REGION Network 4: Start injection
   RUNG wire#powerrail
      { S7_Templates := "SrcType := UInt" } EQ_Contact(in1 := #Current_machine_state, in2 := #st_running_molding_sub3)
      wire#w1
      { S7_Templates := "SrcType := UInt" } EQ_Contact(in1 := #Product_no, in2 := 5)
      Move(in := #container_05gr, out1 => #injection_value)
   END_RUNG
   RUNG wire#w1
      { S7_Templates := "SrcType := UInt" } EQ_Contact(in1 := #Product_no, in2 := 1)
      Move(in := #container_1gr, out1 => #injection_value)
   END_RUNG
   RUNG wire#w1
      { S7_Templates := "SrcType := UInt" } EQ_Contact(in1 := #Product_no, in2 := 2)
      Move(in := #container_2gr, out1 => #injection_value)
   END_RUNG
   RUNG wire#w1
      S_Coil( #Injection_start )
   END_RUNG
   RUNG wire#w1
      Contact( #Injection_start )
      { S7_Templates := "SrcType := Real" } LE_Contact(in1 := #injected_value, in2 := #injection_value)
      wire#w2
      { S7_Templates := "SrcType := Real" } Add(in1 := #injected_value, in2 := 1.03, out => #injected_value)
   END_RUNG
   RUNG wire#w2
      Sub(in1 := #Analog_Inputs.Material_ActLevel, in2 := 0.00103, out => #Analog_Inputs.Material_ActLevel)
   END_RUNG
   RUNG wire#w1
      { S7_Templates := "SrcType := Real" } GT_Contact(in1 := #injected_value, in2 := #injection_value)
      wire#w3
      R_Coil( #Injection_start )
   END_RUNG
   RUNG wire#w3
      "FC_change_machineState"(stop_request := #stop_request, new_stateNo := #st_running_molding_sub4, new_stateDescription := 'Waiting for melting', act_error_code := 0, act_warning_code := 0, act_stateNo => #Current_machine_state, info_actStateNo => #StationInfo.StateNo, info_actStateDescription => #StationInfo.StateDescription, info_errorCode => #StationInfo.ErrorCode, info_warningCode => #StationInfo.WarningCode)
   END_RUNG
   // the same network as SCL:
   #_w1 := #Current_machine_state = #st_running_molding_sub3;
   IF #_w1 AND (#Product_no = 5) THEN #injection_value := #container_05gr; END_IF;
   IF #_w1 AND (#Product_no = 1) THEN #injection_value := #container_1gr; END_IF;
   IF #_w1 AND (#Product_no = 2) THEN #injection_value := #container_2gr; END_IF;
   IF #_w1 THEN #Injection_start := TRUE; END_IF;
   #_w2 := #_w1 AND #Injection_start AND (#injected_value <= #injection_value);
   IF #_w2 THEN
       #injected_value := #injected_value + 1.03;
       #Analog_Inputs.Material_ActLevel := #Analog_Inputs.Material_ActLevel - 0.00103;
   END_IF;
   IF #_w1 AND (#injected_value > #injection_value) THEN
       #Injection_start := FALSE;
       "FC_change_machineState"(stop_request := #stop_request,
                               new_stateNo := #st_running_molding_sub4,
                               new_stateDescription := 'Waiting for melting',
                               act_error_code := 0,
                               act_warning_code := 0,
                               act_stateNo => #Current_machine_state,
                               info_actStateNo => #StationInfo.StateNo,
                               info_actStateDescription => #StationInfo.StateDescription,
                               info_errorCode => #StationInfo.ErrorCode,
                               info_warningCode => #StationInfo.WarningCode);
   END_IF;
END_REGION

REGION Network 5
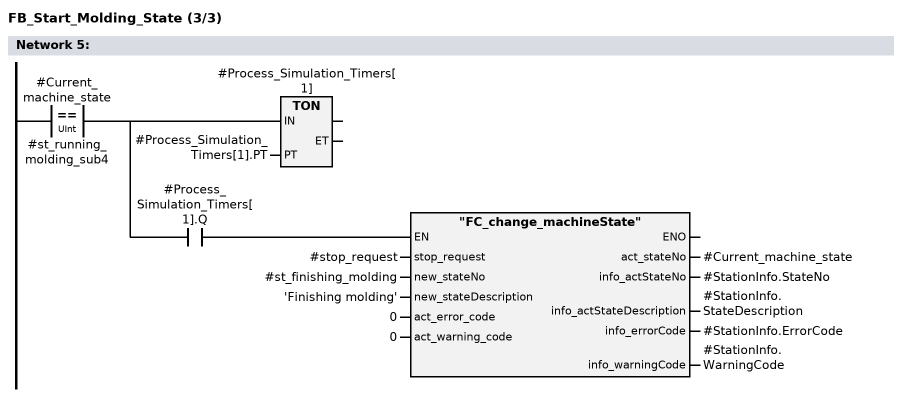
   #_w1 := #Current_machine_state = #st_running_molding_sub4;
   #Process_Simulation_Timers[1].TON(IN := #_w1, PT := #Process_Simulation_Timers[1].PT);
   IF #_w1 AND #Process_Simulation_Timers[1].Q THEN
       "FC_change_machineState"(stop_request := #stop_request,
                               new_stateNo := #st_finishing_molding,
                               new_stateDescription := 'Finishing molding',
                               act_error_code := 0,
                               act_warning_code := 0,
                               act_stateNo => #Current_machine_state,
                               info_actStateNo => #StationInfo.StateNo,
                               info_actStateDescription => #StationInfo.StateDescription,
                               info_errorCode => #StationInfo.ErrorCode,
                               info_warningCode => #StationInfo.WarningCode);
   END_IF;
END_REGION
END_FUNCTION_BLOCK

// folder: Flow4_Finishing_Molding_State

FUNCTION_BLOCK "FB_Finishing_Molding"   // FB12, LAD
{ S7_Optimized_Access := 'TRUE' }
VERSION : 0.1
   VAR_INPUT
      Analog_Inputs : Struct
         Material_ActLevel : Real;
         Temperature_ActLevel : Real;
         Air_Pressure_ActLevel : Real;
         AI_unused1 : Real;
         AI_unused2 : Real;
      END_STRUCT;
      Station_Parameters : Struct
         Hopper : Struct
            ErrorLimit : Real := 1250.0;
            HighLimit : Real := 1000.0;
            LowLimit : Real := 350.0;
            EmptyLimit : Real := 50.0;
         END_STRUCT;
         Temperature : Struct
            ErrorLimit : Real := 600.0;
            HighLimit : Real := 550.0;
            LowLimit : Real := 400.0;
         END_STRUCT;
         Pressure : Struct
            ErrorLimit : Real := 15.0;
            HighLimit : Real := 13.0;
            LowLimit : Real := 10.0;
         END_STRUCT;
         Timeout : Struct
            Mold : Struct
               Open : Time;
               Close : Time;
            END_STRUCT;
            Ejector : Struct
               Open : Time;
               Close : Time;
            END_STRUCT;
            ProductDetect : Time;
            Transfer : Time;
         END_STRUCT;
      END_STRUCT;
   END_VAR
   VAR_OUTPUT
      Ejector_Forward : Bool;
      Ejector_Backward : Bool;
   END_VAR
   VAR_IN_OUT
      Digital_Inputs : Struct
         Start_Button : Bool;
         Stop_Button : Bool;
         Emergency_Stop : Bool;
         Mold_isClosed : Bool;
         Mold_isOpen : Bool;
         Ejector_is_atHome : Bool;
         Ejector_isExtended : Bool;
         Product_Ejected : Bool;
         NextStation_Buffer_Full : Bool;
         DI_unused1 : Bool;
         DI_unused2 : Bool;
         DI_unused3 : Bool;
         DI_unused4 : Bool;
         DI_unused5 : Bool;
         DI_unused6 : Bool;
         DI_unused7 : Bool;
      END_STRUCT;
      stop_request : Bool;
      Current_machine_state : UInt;
      StationInfo : Struct
         StateNo : UInt;
         StateDescription : String;
         ErrorCode : UInt;
         ErrorDescription : String;
         WarningCode : UInt;
         WarninDescription : String;
         TotalProductionTime : Time;
         ProducedCount : UInt;
         OrderCompleted : Bool;
      END_STRUCT;
      Cooler_enable : Bool;
      Mold_open : Bool;
   END_VAR
   VAR
      temp_state : UInt;
      Timeout : Array[0..5] of IEC_TIMER;
      Process_Simulation_Timers : Array[0..20] of IEC_TIMER;
      aux_var1 : Bool;
      deneme_count : IEC_COUNTER;
   END_VAR
   VAR CONSTANT
      st_idle : UInt := 0;
      st_finishing_molding : UInt := 400;
      st_finishing_molding_sub1 : UInt := 401;
      st_finishing_molding_sub2 : UInt := 402;
      st_finishing_molding_sub3 : UInt := 403;
      st_finishing_molding_sub4 : UInt := 404;
      st_finishing_molding_sub5 : UInt := 405;
      st_finishing_molding_sub6 : UInt := 406;
      st_finishing_molding_sub7 : UInt := 407;
      st_finishing_molding_sub8 : UInt := 408;
      st_finishing_molding_sub9 : UInt := 409;
      st_cycle_completed : UInt := 500;
   END_VAR
   VAR_TEMP   // added for the SCL form of the ladder/FBD networks
      _w1 : Bool;
   END_VAR
   // Process_Simulation_Timers[0].PT := T#2S_500MS;
   // Process_Simulation_Timers[1].PT := T#2S_500MS;
   // Process_Simulation_Timers[2].PT := T#500MS;
   // Process_Simulation_Timers[3].PT := T#5S;
   // Process_Simulation_Timers[4].PT := T#10S;
   // Process_Simulation_Timers[10].PT := T#5S;
   // deneme_count.PV := 10;
BEGIN

REGION Network 1
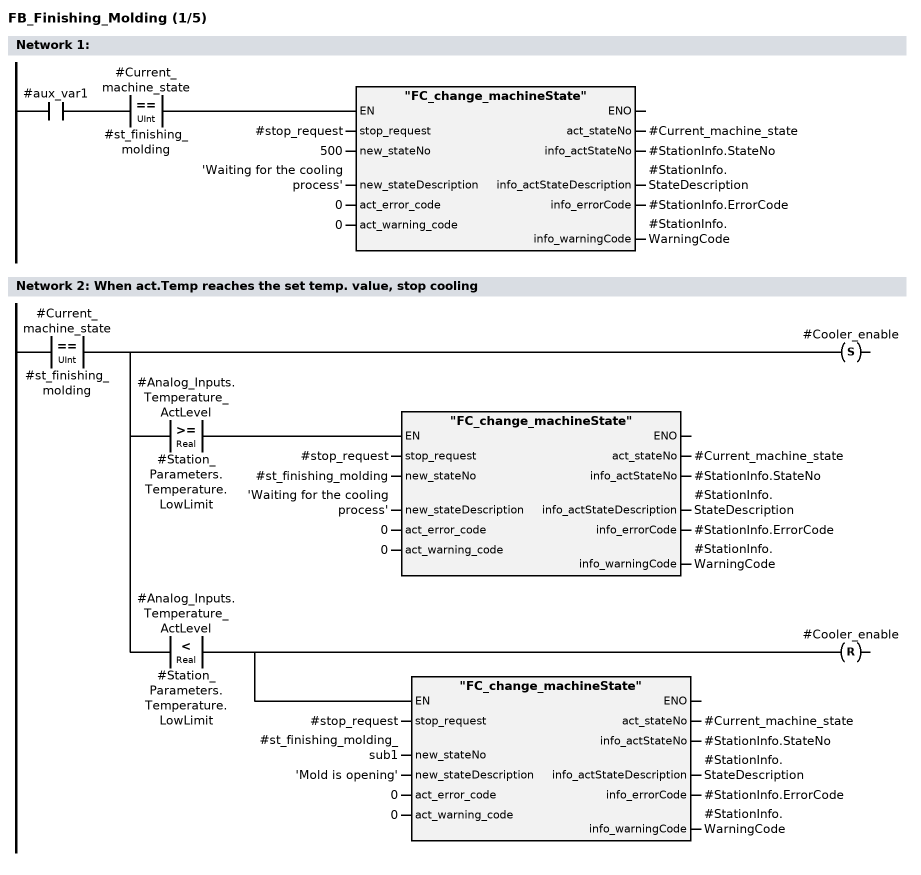
   RUNG wire#powerrail
      Contact( #aux_var1 )
      { S7_Templates := "SrcType := UInt" } EQ_Contact(in1 := #Current_machine_state, in2 := #st_finishing_molding)
      "FC_change_machineState"(stop_request := #stop_request, new_stateNo := 500, new_stateDescription := 'Waiting for the cooling process', act_error_code := 0, act_warning_code := 0, act_stateNo => #Current_machine_state, info_actStateNo => #StationInfo.StateNo, info_actStateDescription => #StationInfo.StateDescription, info_errorCode => #StationInfo.ErrorCode, info_warningCode => #StationInfo.WarningCode)
   END_RUNG
   // the same network as SCL:
   IF #aux_var1 AND (#Current_machine_state = #st_finishing_molding) THEN
       "FC_change_machineState"(stop_request := #stop_request,
                               new_stateNo := 500,
                               new_stateDescription := 'Waiting for the cooling process',
                               act_error_code := 0,
                               act_warning_code := 0,
                               act_stateNo => #Current_machine_state,
                               info_actStateNo => #StationInfo.StateNo,
                               info_actStateDescription => #StationInfo.StateDescription,
                               info_errorCode => #StationInfo.ErrorCode,
                               info_warningCode => #StationInfo.WarningCode);
   END_IF;
END_REGION

REGION Network 2: When act.Temp reaches the set temp. value, stop cooling
   RUNG wire#powerrail
      { S7_Templates := "SrcType := UInt" } EQ_Contact(in1 := #Current_machine_state, in2 := #st_finishing_molding)
      wire#w1
      S_Coil( #Cooler_enable )
   END_RUNG
   RUNG wire#w1
      { S7_Templates := "SrcType := Real" } GE_Contact(in1 := #Analog_Inputs.Temperature_ActLevel, in2 := #Station_Parameters.Temperature.LowLimit)
      "FC_change_machineState"(stop_request := #stop_request, new_stateNo := #st_finishing_molding, new_stateDescription := 'Waiting for the cooling process', act_error_code := 0, act_warning_code := 0, act_stateNo => #Current_machine_state, info_actStateNo => #StationInfo.StateNo, info_actStateDescription => #StationInfo.StateDescription, info_errorCode => #StationInfo.ErrorCode, info_warningCode => #StationInfo.WarningCode)
   END_RUNG
   RUNG wire#w1
      { S7_Templates := "SrcType := Real" } LT_Contact(in1 := #Analog_Inputs.Temperature_ActLevel, in2 := #Station_Parameters.Temperature.LowLimit)
      wire#w2
      R_Coil( #Cooler_enable )
   END_RUNG
   RUNG wire#w2
      "FC_change_machineState"(stop_request := #stop_request, new_stateNo := #st_finishing_molding_sub1, new_stateDescription := 'Mold is opening', act_error_code := 0, act_warning_code := 0, act_stateNo => #Current_machine_state, info_actStateNo => #StationInfo.StateNo, info_actStateDescription => #StationInfo.StateDescription, info_errorCode => #StationInfo.ErrorCode, info_warningCode => #StationInfo.WarningCode)
   END_RUNG
   // the same network as SCL:
   #_w1 := #Current_machine_state = #st_finishing_molding;
   IF #_w1 THEN #Cooler_enable := TRUE; END_IF;
   IF #_w1 AND (#Analog_Inputs.Temperature_ActLevel >= #Station_Parameters.Temperature.LowLimit) THEN
       "FC_change_machineState"(stop_request := #stop_request,
                               new_stateNo := #st_finishing_molding,
                               new_stateDescription := 'Waiting for the cooling process',
                               act_error_code := 0,
                               act_warning_code := 0,
                               act_stateNo => #Current_machine_state,
                               info_actStateNo => #StationInfo.StateNo,
                               info_actStateDescription => #StationInfo.StateDescription,
                               info_errorCode => #StationInfo.ErrorCode,
                               info_warningCode => #StationInfo.WarningCode);
   END_IF;
   IF #_w1 AND (#Analog_Inputs.Temperature_ActLevel < #Station_Parameters.Temperature.LowLimit) THEN
       #Cooler_enable := FALSE;
       "FC_change_machineState"(stop_request := #stop_request,
                               new_stateNo := #st_finishing_molding_sub1,
                               new_stateDescription := 'Mold is opening',
                               act_error_code := 0,
                               act_warning_code := 0,
                               act_stateNo => #Current_machine_state,
                               info_actStateNo => #StationInfo.StateNo,
                               info_actStateDescription => #StationInfo.StateDescription,
                               info_errorCode => #StationInfo.ErrorCode,
                               info_warningCode => #StationInfo.WarningCode);
   END_IF;
END_REGION

REGION Network 3: Open the mold
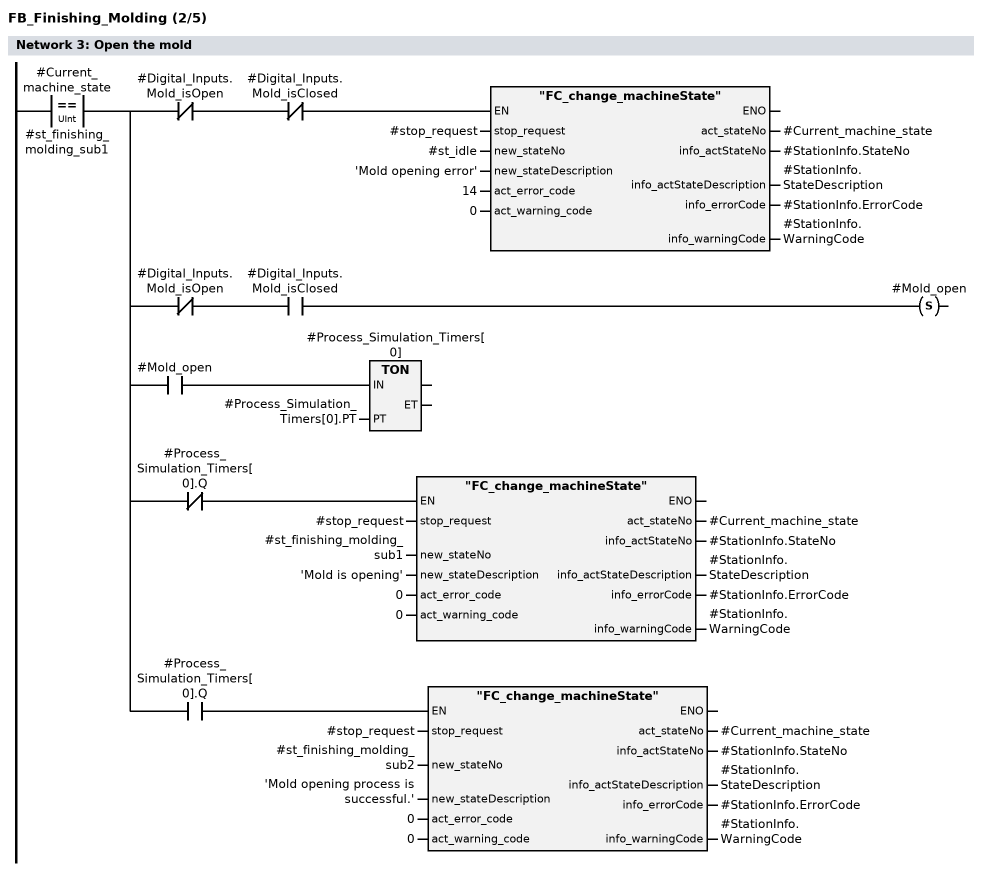
   #_w1 := #Current_machine_state = #st_finishing_molding_sub1;
   IF #_w1 AND NOT #Digital_Inputs.Mold_isOpen AND NOT #Digital_Inputs.Mold_isClosed THEN
       "FC_change_machineState"(stop_request := #stop_request,
                               new_stateNo := #st_idle,
                               new_stateDescription := 'Mold opening error',
                               act_error_code := 14,
                               act_warning_code := 0,
                               act_stateNo => #Current_machine_state,
                               info_actStateNo => #StationInfo.StateNo,
                               info_actStateDescription => #StationInfo.StateDescription,
                               info_errorCode => #StationInfo.ErrorCode,
                               info_warningCode => #StationInfo.WarningCode);
   END_IF;
   IF #_w1 AND NOT #Digital_Inputs.Mold_isOpen AND #Digital_Inputs.Mold_isClosed THEN
       #Mold_open := TRUE;
   END_IF;
   #Process_Simulation_Timers[0].TON(IN := #_w1 AND #Mold_open, PT := #Process_Simulation_Timers[0].PT);
   IF #_w1 AND NOT #Process_Simulation_Timers[0].Q THEN
       "FC_change_machineState"(stop_request := #stop_request,
                               new_stateNo := #st_finishing_molding_sub1,
                               new_stateDescription := 'Mold is opening',
                               act_error_code := 0,
                               act_warning_code := 0,
                               act_stateNo => #Current_machine_state,
                               info_actStateNo => #StationInfo.StateNo,
                               info_actStateDescription => #StationInfo.StateDescription,
                               info_errorCode => #StationInfo.ErrorCode,
                               info_warningCode => #StationInfo.WarningCode);
   END_IF;
   IF #_w1 AND #Process_Simulation_Timers[0].Q THEN
       "FC_change_machineState"(stop_request := #stop_request,
                               new_stateNo := #st_finishing_molding_sub2,
                               new_stateDescription := 'Mold opening process is successful.',
                               act_error_code := 0,
                               act_warning_code := 0,
                               act_stateNo => #Current_machine_state,
                               info_actStateNo => #StationInfo.StateNo,
                               info_actStateDescription => #StationInfo.StateDescription,
                               info_errorCode => #StationInfo.ErrorCode,
                               info_warningCode => #StationInfo.WarningCode);
   END_IF;
END_REGION

REGION Network 4: Start Ejection
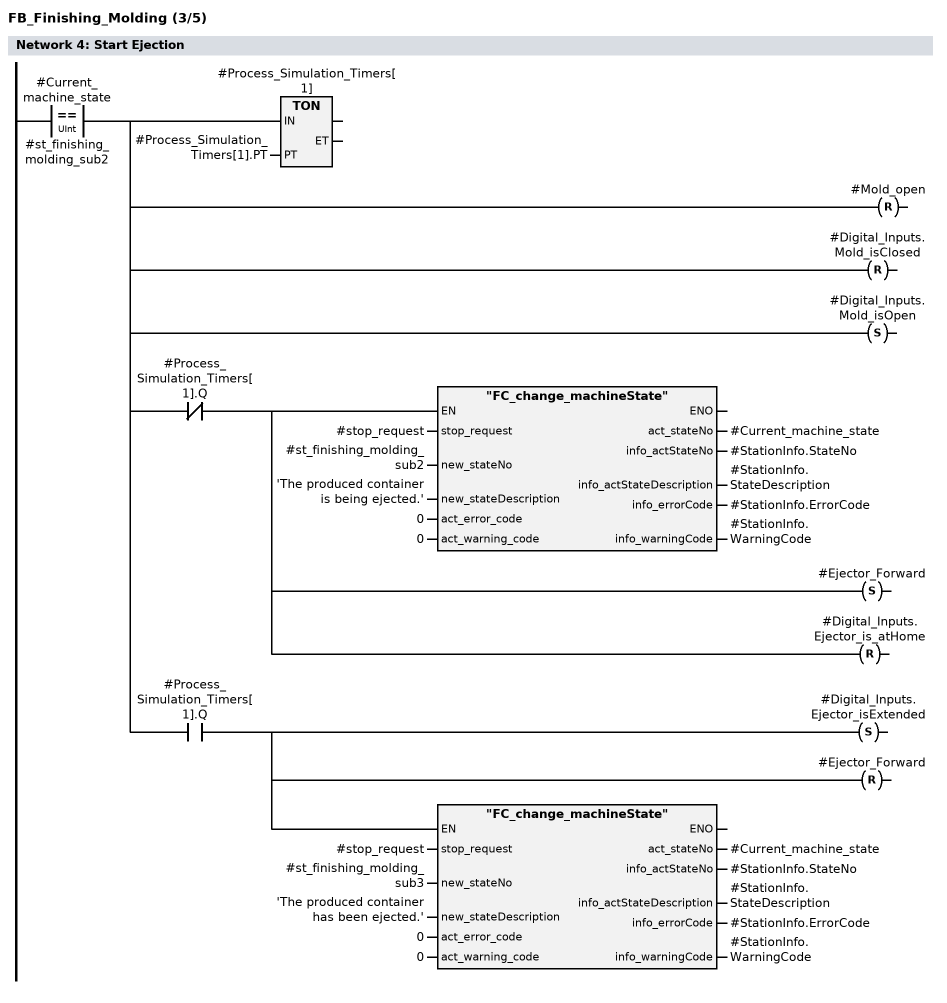
   #_w1 := #Current_machine_state = #st_finishing_molding_sub2;
   #Process_Simulation_Timers[1].TON(IN := #_w1, PT := #Process_Simulation_Timers[1].PT);
   IF #_w1 THEN
       #Mold_open := FALSE;
       #Digital_Inputs.Mold_isClosed := FALSE;
       #Digital_Inputs.Mold_isOpen := TRUE;
   END_IF;
   IF #_w1 AND NOT #Process_Simulation_Timers[1].Q THEN
       "FC_change_machineState"(stop_request := #stop_request,
                               new_stateNo := #st_finishing_molding_sub2,
                               new_stateDescription := 'The produced container is being ejected.',
                               act_error_code := 0,
                               act_warning_code := 0,
                               act_stateNo => #Current_machine_state,
                               info_actStateNo => #StationInfo.StateNo,
                               info_actStateDescription => #StationInfo.StateDescription,
                               info_errorCode => #StationInfo.ErrorCode,
                               info_warningCode => #StationInfo.WarningCode);
       #Ejector_Forward := TRUE;
       #Digital_Inputs.Ejector_is_atHome := FALSE;
   END_IF;
   IF #_w1 AND #Process_Simulation_Timers[1].Q THEN
       #Digital_Inputs.Ejector_isExtended := TRUE;
       #Ejector_Forward := FALSE;
       "FC_change_machineState"(stop_request := #stop_request,
                               new_stateNo := #st_finishing_molding_sub3,
                               new_stateDescription := 'The produced container has been ejected.',
                               act_error_code := 0,
                               act_warning_code := 0,
                               act_stateNo => #Current_machine_state,
                               info_actStateNo => #StationInfo.StateNo,
                               info_actStateDescription => #StationInfo.StateDescription,
                               info_errorCode => #StationInfo.ErrorCode,
                               info_warningCode => #StationInfo.WarningCode);
   END_IF;
END_REGION

REGION Network 5: Stop Ejection
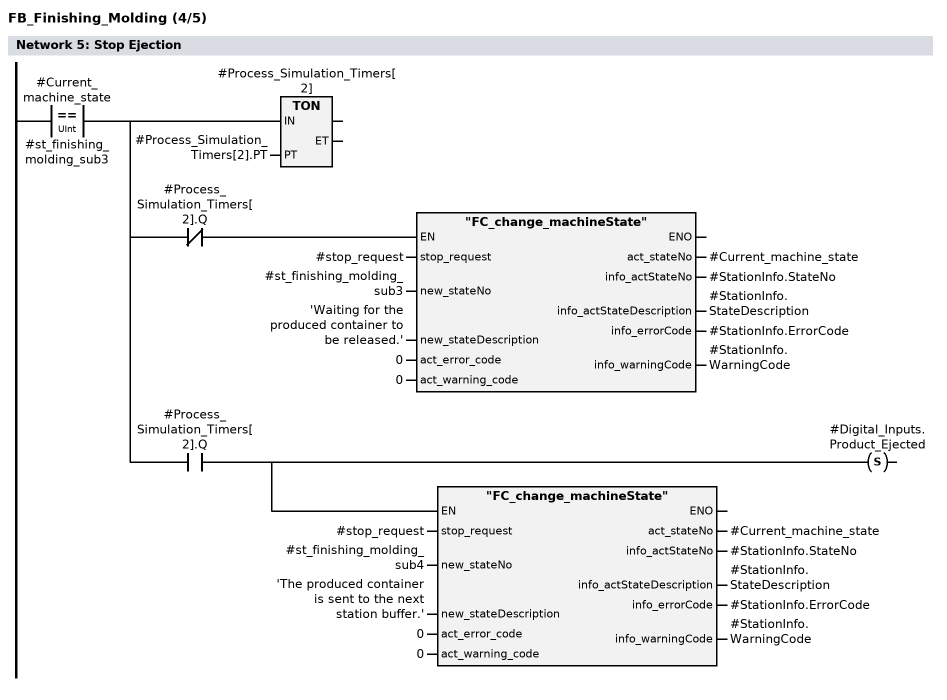
   #_w1 := #Current_machine_state = #st_finishing_molding_sub3;
   #Process_Simulation_Timers[2].TON(IN := #_w1, PT := #Process_Simulation_Timers[2].PT);
   IF #_w1 AND NOT #Process_Simulation_Timers[2].Q THEN
       "FC_change_machineState"(stop_request := #stop_request,
                               new_stateNo := #st_finishing_molding_sub3,
                               new_stateDescription := 'Waiting for the produced container to be released.',
                               act_error_code := 0,
                               act_warning_code := 0,
                               act_stateNo => #Current_machine_state,
                               info_actStateNo => #StationInfo.StateNo,
                               info_actStateDescription => #StationInfo.StateDescription,
                               info_errorCode => #StationInfo.ErrorCode,
                               info_warningCode => #StationInfo.WarningCode);
   END_IF;
   IF #_w1 AND #Process_Simulation_Timers[2].Q THEN
       #Digital_Inputs.Product_Ejected := TRUE;
       "FC_change_machineState"(stop_request := #stop_request,
                               new_stateNo := #st_finishing_molding_sub4,
                               new_stateDescription := 'The produced container is sent to the next station buffer.',
                               act_error_code := 0,
                               act_warning_code := 0,
                               act_stateNo => #Current_machine_state,
                               info_actStateNo => #StationInfo.StateNo,
                               info_actStateDescription => #StationInfo.StateDescription,
                               info_errorCode => #StationInfo.ErrorCode,
                               info_warningCode => #StationInfo.WarningCode);
   END_IF;
END_REGION

REGION Network 6: Send to the next station
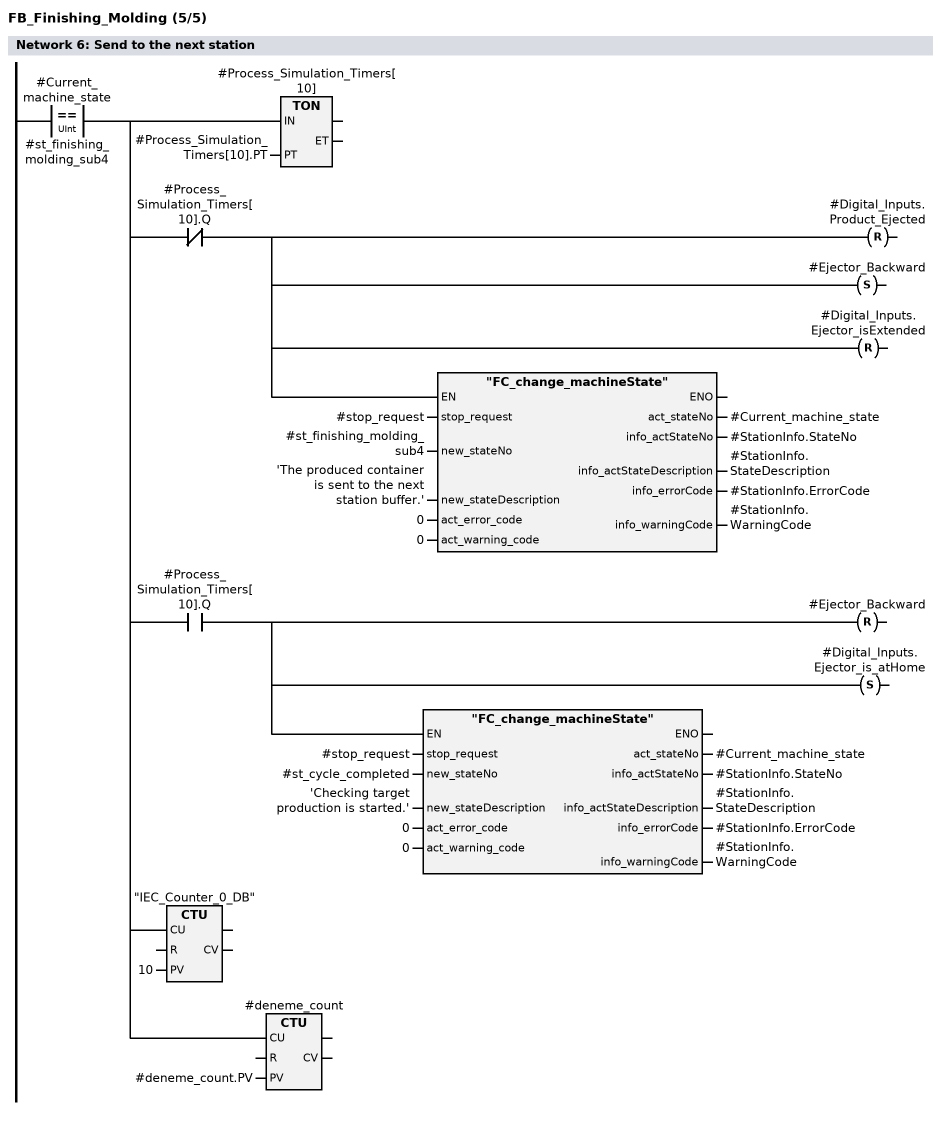
   #_w1 := #Current_machine_state = #st_finishing_molding_sub4;
   #Process_Simulation_Timers[10].TON(IN := #_w1, PT := #Process_Simulation_Timers[10].PT);
   IF #_w1 AND NOT #Process_Simulation_Timers[10].Q THEN
       #Digital_Inputs.Product_Ejected := FALSE;
       #Ejector_Backward := TRUE;
       #Digital_Inputs.Ejector_isExtended := FALSE;
       "FC_change_machineState"(stop_request := #stop_request,
                               new_stateNo := #st_finishing_molding_sub4,
                               new_stateDescription := 'The produced container is sent to the next station buffer.',
                               act_error_code := 0,
                               act_warning_code := 0,
                               act_stateNo => #Current_machine_state,
                               info_actStateNo => #StationInfo.StateNo,
                               info_actStateDescription => #StationInfo.StateDescription,
                               info_errorCode => #StationInfo.ErrorCode,
                               info_warningCode => #StationInfo.WarningCode);
   END_IF;
   IF #_w1 AND #Process_Simulation_Timers[10].Q THEN
       #Ejector_Backward := FALSE;
       #Digital_Inputs.Ejector_is_atHome := TRUE;
       "FC_change_machineState"(stop_request := #stop_request,
                               new_stateNo := #st_cycle_completed,
                               new_stateDescription := 'Checking target production is started.',
                               act_error_code := 0,
                               act_warning_code := 0,
                               act_stateNo => #Current_machine_state,
                               info_actStateNo => #StationInfo.StateNo,
                               info_actStateDescription => #StationInfo.StateDescription,
                               info_errorCode => #StationInfo.ErrorCode,
                               info_warningCode => #StationInfo.WarningCode);
   END_IF;
   "IEC_Counter_0_DB".CTU(CU := #_w1, PV := 10);
   #deneme_count.CTU(CU := #_w1, PV := #deneme_count.PV);
END_REGION
END_FUNCTION_BLOCK

// folder: Flow5_Checking_Target_Production

FUNCTION_BLOCK "FB_Checking_Target_Production"   // FB11, LAD
{ S7_Optimized_Access := 'TRUE' }
VERSION : 0.1
   VAR_INPUT
      target_quantity : UInt;
   END_VAR
   VAR_IN_OUT
      stop_request : Bool;
      Current_machine_state : UInt;
      StationInfo : Struct
         StateNo : UInt;
         StateDescription : String;
         ErrorCode : UInt;
         ErrorDescription : String;
         WarningCode : UInt;
         WarninDescription : String;
         TotalProductionTime : Time;
         ProducedCount : UInt;
         OrderCompleted : Bool;
      END_STRUCT;
   END_VAR
   VAR
      Timeout : Array[0..5] of IEC_TIMER;
      Process_Simulation_Timers : Array[0..20] of IEC_TIMER;
      Production_Counter : Array[0..10] of IEC_UCOUNTER;
      aux_var1 : Bool;
   END_VAR
   VAR_TEMP
      cycle_completed : Bool;
      continue : Bool;
   END_VAR
   VAR CONSTANT
      st_idle : UInt := 0;
      st_cycle_completed : UInt := 500;
      st_cycle_completed_sub1 : UInt := 501;
      st_cycle_completed_sub2 : UInt := 502;
      st_cycle_completed_sub3 : UInt := 503;
      st_cycle_completed_sub4 : UInt := 504;
      st_cycle_completed_sub5 : UInt := 505;
      st_cycle_completed_sub6 : UInt := 506;
      st_cycle_completed_sub7 : UInt := 507;
      st_cycle_completed_sub8 : UInt := 508;
      st_cycle_completed_sub9 : UInt := 509;
      st_checking_order_target : UInt := 600;
      st_checking_initial_safety : UInt := 200;
      st_order_finishing : UInt := 700;
      st_checking_order_sub2 : UInt := 102;
   END_VAR
   VAR_TEMP   // added for the SCL form of the ladder/FBD networks
      _w1 : Bool;
   END_VAR
   // Process_Simulation_Timers[0].PT := T#3S;
   // Process_Simulation_Timers[1].PT := T#4S;
   // Process_Simulation_Timers[2].PT := T#10S;
   // Process_Simulation_Timers[3].PT := T#3S;
BEGIN

REGION Network 1: Check target production
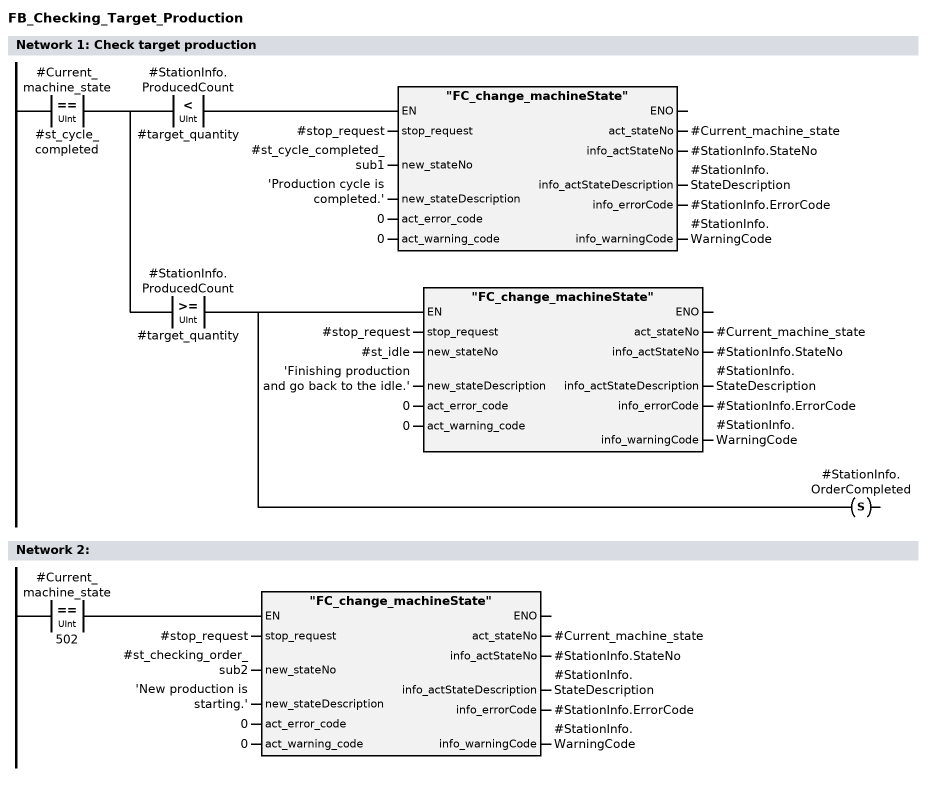
   RUNG wire#powerrail
      { S7_Templates := "SrcType := UInt" } EQ_Contact(in1 := #Current_machine_state, in2 := #st_cycle_completed)
      wire#w1
      { S7_Templates := "SrcType := UInt" } LT_Contact(in1 := #StationInfo.ProducedCount, in2 := #target_quantity)
      "FC_change_machineState"(stop_request := #stop_request, new_stateNo := #st_cycle_completed_sub1, new_stateDescription := 'Production cycle is completed.', act_error_code := 0, act_warning_code := 0, act_stateNo => #Current_machine_state, info_actStateNo => #StationInfo.StateNo, info_actStateDescription => #StationInfo.StateDescription, info_errorCode => #StationInfo.ErrorCode, info_warningCode => #StationInfo.WarningCode)
   END_RUNG
   RUNG wire#w1
      { S7_Templates := "SrcType := UInt" } GE_Contact(in1 := #StationInfo.ProducedCount, in2 := #target_quantity)
      wire#w2
      "FC_change_machineState"(stop_request := #stop_request, new_stateNo := #st_idle, new_stateDescription := 'Finishing production and go back to the idle.', act_error_code := 0, act_warning_code := 0, act_stateNo => #Current_machine_state, info_actStateNo => #StationInfo.StateNo, info_actStateDescription => #StationInfo.StateDescription, info_errorCode => #StationInfo.ErrorCode, info_warningCode => #StationInfo.WarningCode)
   END_RUNG
   RUNG wire#w2
      S_Coil( #StationInfo.OrderCompleted )
   END_RUNG
   // the same network as SCL:
   #_w1 := #Current_machine_state = #st_cycle_completed;
   IF #_w1 AND (#StationInfo.ProducedCount < #target_quantity) THEN
       "FC_change_machineState"(stop_request := #stop_request,
                               new_stateNo := #st_cycle_completed_sub1,
                               new_stateDescription := 'Production cycle is completed.',
                               act_error_code := 0,
                               act_warning_code := 0,
                               act_stateNo => #Current_machine_state,
                               info_actStateNo => #StationInfo.StateNo,
                               info_actStateDescription => #StationInfo.StateDescription,
                               info_errorCode => #StationInfo.ErrorCode,
                               info_warningCode => #StationInfo.WarningCode);
   END_IF;
   IF #_w1 AND (#StationInfo.ProducedCount >= #target_quantity) THEN
       "FC_change_machineState"(stop_request := #stop_request,
                               new_stateNo := #st_idle,
                               new_stateDescription := 'Finishing production and go back to the idle.',
                               act_error_code := 0,
                               act_warning_code := 0,
                               act_stateNo => #Current_machine_state,
                               info_actStateNo => #StationInfo.StateNo,
                               info_actStateDescription => #StationInfo.StateDescription,
                               info_errorCode => #StationInfo.ErrorCode,
                               info_warningCode => #StationInfo.WarningCode);
       #StationInfo.OrderCompleted := TRUE;
   END_IF;
END_REGION

REGION Network 2
   RUNG wire#powerrail
      { S7_Templates := "SrcType := UInt" } EQ_Contact(in1 := #Current_machine_state, in2 := 502)
      "FC_change_machineState"(stop_request := #stop_request, new_stateNo := #st_checking_order_sub2, new_stateDescription := 'New production is starting.', act_error_code := 0, act_warning_code := 0, act_stateNo => #Current_machine_state, info_actStateNo => #StationInfo.StateNo, info_actStateDescription => #StationInfo.StateDescription, info_errorCode => #StationInfo.ErrorCode, info_warningCode => #StationInfo.WarningCode)
   END_RUNG
   // the same network as SCL:
   IF #Current_machine_state = 502 THEN
       "FC_change_machineState"(stop_request := #stop_request,
                               new_stateNo := #st_checking_order_sub2,
                               new_stateDescription := 'New production is starting.',
                               act_error_code := 0,
                               act_warning_code := 0,
                               act_stateNo => #Current_machine_state,
                               info_actStateNo => #StationInfo.StateNo,
                               info_actStateDescription => #StationInfo.StateDescription,
                               info_errorCode => #StationInfo.ErrorCode,
                               info_warningCode => #StationInfo.WarningCode);
   END_IF;
END_REGION
END_FUNCTION_BLOCK

// folder: Functions

FUNCTION "FC_get_time_data" : Void   // FC1, LAD
{ S7_Optimized_Access := 'TRUE' }
VERSION : 0.1
   VAR_OUTPUT
      actYear : UInt;
      actMonth : UInt;
      actDay : UInt;
      timeStamp : UDInt;
      errorGettingTime : Int;
   END_VAR
   VAR_TEMP
      timeData : DTL;
      gettingTimeState : Int;
   END_VAR
BEGIN

REGION Network 1
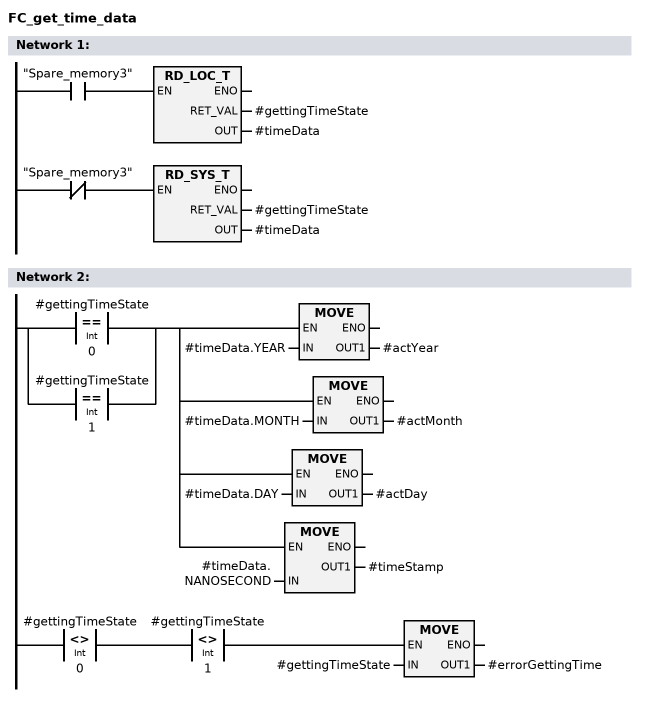
   IF "Spare_memory3" THEN #gettingTimeState := RD_LOC_T(OUT => #timeData); END_IF;
   IF NOT "Spare_memory3" THEN #gettingTimeState := RD_SYS_T(OUT => #timeData); END_IF;
END_REGION

REGION Network 2
   RUNG wire#powerrail
      { S7_Templates := "SrcType := Int" } EQ_Contact(in1 := #gettingTimeState, in2 := 0)
      wire#w1
      Move(in := #timeData.YEAR, out1 => #actYear)
   END_RUNG
   RUNG wire#powerrail
      { S7_Templates := "SrcType := Int" } EQ_Contact(in1 := #gettingTimeState, in2 := 1)
   END_RUNG wire#w1
   RUNG wire#w1
      Move(in := #timeData.MONTH, out1 => #actMonth)
   END_RUNG
   RUNG wire#w1
      Move(in := #timeData.DAY, out1 => #actDay)
   END_RUNG
   RUNG wire#w1
      Move(in := #timeData.NANOSECOND, out1 => #timeStamp)
   END_RUNG
   RUNG wire#powerrail
      { S7_Templates := "SrcType := Int" } NE_Contact(in1 := #gettingTimeState, in2 := 0)
      { S7_Templates := "SrcType := Int" } NE_Contact(in1 := #gettingTimeState, in2 := 1)
      Move(in := #gettingTimeState, out1 => #errorGettingTime)
   END_RUNG
   // the same network as SCL:
   IF (#gettingTimeState = 0) OR (#gettingTimeState = 1) THEN
       #actYear := #timeData.YEAR;
       #actMonth := #timeData.MONTH;
       #actDay := #timeData.DAY;
       #timeStamp := #timeData.NANOSECOND;
   END_IF;
   IF (#gettingTimeState <> 0) AND (#gettingTimeState <> 1) THEN
       #errorGettingTime := #gettingTimeState;
   END_IF;
END_REGION
END_FUNCTION

FUNCTION "FC_change_machineState" : Void   // FC2, LAD
{ S7_Optimized_Access := 'TRUE' }
VERSION : 0.1
   VAR_INPUT
      stop_request : Bool;
      new_stateNo : UInt;
      new_stateDescription : String;
      act_error_code : UInt;
      act_warning_code : UInt;
   END_VAR
   VAR_OUTPUT
      act_stateNo : UInt;
      info_actStateNo : UInt;
      info_actStateDescription : String;
      info_errorCode : UInt;
      info_warningCode : UInt;
   END_VAR
   VAR CONSTANT
      st_idle : UInt := 0;
   END_VAR
BEGIN

REGION Network 1: No Stop Request Received
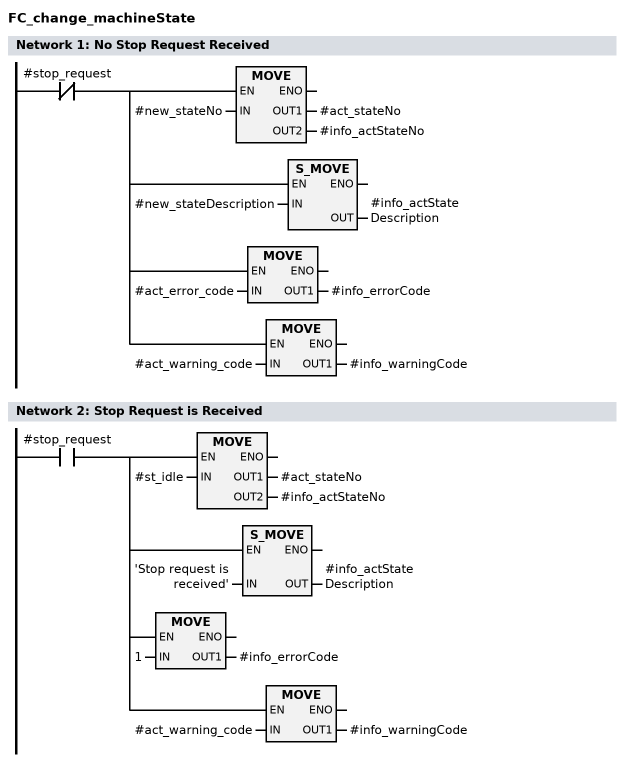
   RUNG wire#powerrail
      I_Contact( #stop_request )
      wire#w1
      Move(in := #new_stateNo, out1 => #act_stateNo, out2 => #info_actStateNo)
   END_RUNG
   RUNG wire#w1
      S_Move(in := #new_stateDescription, out => #info_actStateDescription)
   END_RUNG
   RUNG wire#w1
      Move(in := #act_error_code, out1 => #info_errorCode)
   END_RUNG
   RUNG wire#w1
      Move(in := #act_warning_code, out1 => #info_warningCode)
   END_RUNG
   // the same network as SCL:
   IF NOT #stop_request THEN
       #act_stateNo := #new_stateNo;
       #info_actStateNo := #new_stateNo;
       #info_actStateDescription := #new_stateDescription;
       #info_errorCode := #act_error_code;
       #info_warningCode := #act_warning_code;
   END_IF;
END_REGION

REGION Network 2: Stop Request is Received
   RUNG wire#powerrail
      Contact( #stop_request )
      wire#w1
      Move(in := #st_idle, out1 => #act_stateNo, out2 => #info_actStateNo)
   END_RUNG
   RUNG wire#w1
      S_Move(in := 'Stop request is received', out => #info_actStateDescription)
   END_RUNG
   RUNG wire#w1
      Move(in := 1, out1 => #info_errorCode)
   END_RUNG
   RUNG wire#w1
      Move(in := #act_warning_code, out1 => #info_warningCode)
   END_RUNG
   // the same network as SCL:
   IF #stop_request THEN
       #act_stateNo := #st_idle;
       #info_actStateNo := #st_idle;
       #info_actStateDescription := 'Stop request is received';
       #info_errorCode := 1;
       #info_warningCode := #act_warning_code;
   END_IF;
END_REGION
END_FUNCTION

// folder: Machine_transition

FUNCTION_BLOCK "FB_SubTransition"   // FB3, LAD
{ S7_Optimized_Access := 'TRUE' }
VERSION : 0.1
   VAR_INPUT
      new_state : UInt;
   END_VAR
   VAR_OUTPUT
      new_machine_state : UInt;
      previous_state_done : Bool;
   END_VAR
   VAR_IN_OUT
      stop_request : Bool;
   END_VAR
   VAR CONSTANT
      st_idle : UInt := 0;
   END_VAR
BEGIN

REGION Network 1: No Stop Request
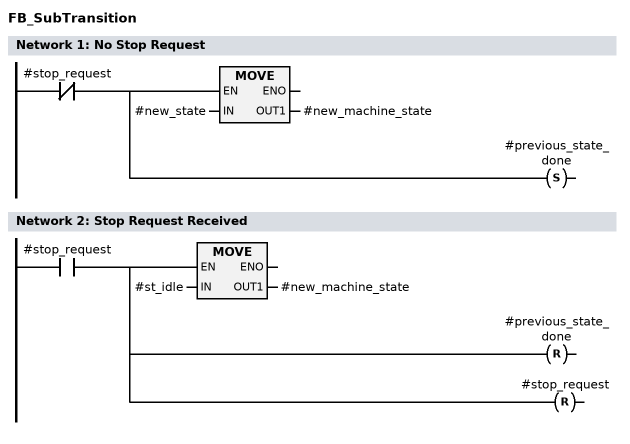
   RUNG wire#powerrail
      I_Contact( #stop_request )
      wire#w1
      Move(in := #new_state, out1 => #new_machine_state)
   END_RUNG
   RUNG wire#w1
      S_Coil( #previous_state_done )
   END_RUNG
   // the same network as SCL:
   IF NOT #stop_request THEN
       #new_machine_state := #new_state;
       #previous_state_done := TRUE;
   END_IF;
END_REGION

REGION Network 2: Stop Request Received
   RUNG wire#powerrail
      Contact( #stop_request )
      wire#w1
      Move(in := #st_idle, out1 => #new_machine_state)
   END_RUNG
   RUNG wire#w1
      R_Coil( #previous_state_done )
   END_RUNG
   RUNG wire#w1
      R_Coil( #stop_request )
   END_RUNG
   // the same network as SCL:
   IF #stop_request THEN
       #new_machine_state := #st_idle;
       #previous_state_done := FALSE;
       #stop_request := FALSE;
   END_IF;
END_REGION
END_FUNCTION_BLOCK

FUNCTION_BLOCK "FB_control_state_transition"   // FB6, LAD
TITLE = This FB sets the machine status
{ S7_Optimized_Access := 'TRUE' }
VERSION : 0.1
   VAR_INPUT
      is_start_btn_activated : Bool;
      is_stop_btn_activated : Bool;
   END_VAR
   VAR_IN_OUT
      current_machine_state : UInt;
      is_previous_state_done : Bool;
   END_VAR
   VAR
      temp_state : UInt;
      initial_temp_state : UInt;
      stop_request : Bool;
   END_VAR
   VAR CONSTANT
      st_idle : UInt := 0;
      st_checking_order : UInt := 10;
      st_checking_initial_safety : UInt := 20;
      st_checking_material_level : UInt := 30;
      st_running_molding : UInt := 40;
      st_finishing_molding : UInt := 50;
      st_cycle_completed : UInt := 60;
      st_checking_order_target : UInt := 70;
      st_order_finishing : UInt := 80;
      st_fault : UInt := 300;
   END_VAR
   VAR_TEMP   // added for the SCL form of the ladder/FBD networks
      _w1 : Bool;
   END_VAR
BEGIN

REGION Network 1: Control Stop Request
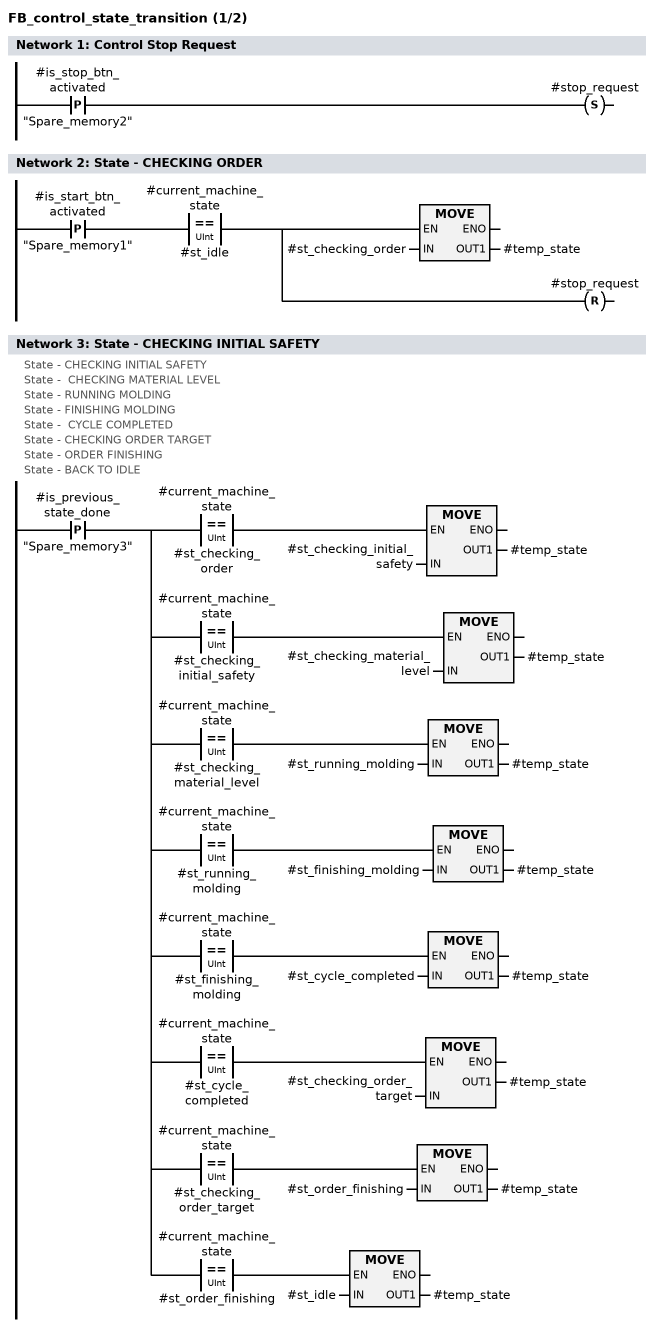
   RUNG wire#powerrail
      P_Contact(operand := #is_stop_btn_activated, bit := "Spare_memory2")
      S_Coil( #stop_request )
   END_RUNG
   // the same network as SCL:
   #_w1 := #is_stop_btn_activated AND NOT "Spare_memory2";   // rising edge of #is_stop_btn_activated
   "Spare_memory2" := #is_stop_btn_activated;
   IF #_w1 THEN #stop_request := TRUE; END_IF;
END_REGION

REGION Network 2: State - CHECKING ORDER
   RUNG wire#powerrail
      P_Contact(operand := #is_start_btn_activated, bit := "Spare_memory1")
      { S7_Templates := "SrcType := UInt" } EQ_Contact(in1 := #current_machine_state, in2 := #st_idle)
      wire#w1
      Move(in := #st_checking_order, out1 => #temp_state)
   END_RUNG
   RUNG wire#w1
      R_Coil( #stop_request )
   END_RUNG
   // the same network as SCL:
   #_w1 := #is_start_btn_activated AND NOT "Spare_memory1";   // rising edge of #is_start_btn_activated
   "Spare_memory1" := #is_start_btn_activated;
   IF #_w1 AND (#current_machine_state = #st_idle) THEN
       #temp_state := #st_checking_order;
       #stop_request := FALSE;
   END_IF;
END_REGION

REGION Network 3: State - CHECKING INITIAL SAFETY
   // State - CHECKING INITIAL SAFETY
   // State -  CHECKING MATERIAL LEVEL
   // State - RUNNING MOLDING
   // State - FINISHING MOLDING
   // State -  CYCLE COMPLETED
   // State - CHECKING ORDER TARGET
   // State - ORDER FINISHING 
   // State - BACK TO IDLE
   RUNG wire#powerrail
      P_Contact(operand := #is_previous_state_done, bit := "Spare_memory3")
      wire#w1
      { S7_Templates := "SrcType := UInt" } EQ_Contact(in1 := #current_machine_state, in2 := #st_checking_order)
      Move(in := #st_checking_initial_safety, out1 => #temp_state)
   END_RUNG
   RUNG wire#w1
      { S7_Templates := "SrcType := UInt" } EQ_Contact(in1 := #current_machine_state, in2 := #st_checking_initial_safety)
      Move(in := #st_checking_material_level, out1 => #temp_state)
   END_RUNG
   RUNG wire#w1
      { S7_Templates := "SrcType := UInt" } EQ_Contact(in1 := #current_machine_state, in2 := #st_checking_material_level)
      Move(in := #st_running_molding, out1 => #temp_state)
   END_RUNG
   RUNG wire#w1
      { S7_Templates := "SrcType := UInt" } EQ_Contact(in1 := #current_machine_state, in2 := #st_running_molding)
      Move(in := #st_finishing_molding, out1 => #temp_state)
   END_RUNG
   RUNG wire#w1
      { S7_Templates := "SrcType := UInt" } EQ_Contact(in1 := #current_machine_state, in2 := #st_finishing_molding)
      Move(in := #st_cycle_completed, out1 => #temp_state)
   END_RUNG
   RUNG wire#w1
      { S7_Templates := "SrcType := UInt" } EQ_Contact(in1 := #current_machine_state, in2 := #st_cycle_completed)
      Move(in := #st_checking_order_target, out1 => #temp_state)
   END_RUNG
   RUNG wire#w1
      { S7_Templates := "SrcType := UInt" } EQ_Contact(in1 := #current_machine_state, in2 := #st_checking_order_target)
      Move(in := #st_order_finishing, out1 => #temp_state)
   END_RUNG
   RUNG wire#w1
      { S7_Templates := "SrcType := UInt" } EQ_Contact(in1 := #current_machine_state, in2 := #st_order_finishing)
      Move(in := #st_idle, out1 => #temp_state)
   END_RUNG
   // the same network as SCL:
   #_w1 := #is_previous_state_done AND NOT "Spare_memory3";   // rising edge of #is_previous_state_done
   "Spare_memory3" := #is_previous_state_done;
   IF #_w1 AND (#current_machine_state = #st_checking_order) THEN
       #temp_state := #st_checking_initial_safety;
   END_IF;
   IF #_w1 AND (#current_machine_state = #st_checking_initial_safety) THEN
       #temp_state := #st_checking_material_level;
   END_IF;
   IF #_w1 AND (#current_machine_state = #st_checking_material_level) THEN
       #temp_state := #st_running_molding;
   END_IF;
   IF #_w1 AND (#current_machine_state = #st_running_molding) THEN
       #temp_state := #st_finishing_molding;
   END_IF;
   IF #_w1 AND (#current_machine_state = #st_finishing_molding) THEN
       #temp_state := #st_cycle_completed;
   END_IF;
   IF #_w1 AND (#current_machine_state = #st_cycle_completed) THEN
       #temp_state := #st_checking_order_target;
   END_IF;
   IF #_w1 AND (#current_machine_state = #st_checking_order_target) THEN
       #temp_state := #st_order_finishing;
   END_IF;
   IF #_w1 AND (#current_machine_state = #st_order_finishing) THEN #temp_state := #st_idle; END_IF;
END_REGION

REGION Network 4: Set the current machine state to new state value
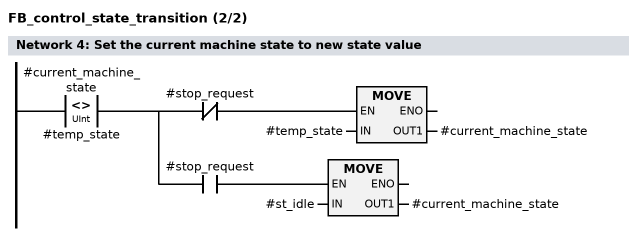
   RUNG wire#powerrail
      { S7_Templates := "SrcType := UInt" } NE_Contact(in1 := #current_machine_state, in2 := #temp_state)
      wire#w1
      I_Contact( #stop_request )
      Move(in := #temp_state, out1 => #current_machine_state)
   END_RUNG
   RUNG wire#w1
      Contact( #stop_request )
      Move(in := #st_idle, out1 => #current_machine_state)
   END_RUNG
   // the same network as SCL:
   #_w1 := #current_machine_state <> #temp_state;
   IF #_w1 AND NOT #stop_request THEN #current_machine_state := #temp_state; END_IF;
   IF #_w1 AND #stop_request THEN #current_machine_state := #st_idle; END_IF;
END_REGION
END_FUNCTION_BLOCK

// folder: Manage_outputs

FUNCTION_BLOCK "FB_manage_outputs"   // FB8, LAD
{ S7_Optimized_Access := 'TRUE' }
VERSION : 0.1
BEGIN

REGION Network 1: Feeder_Start
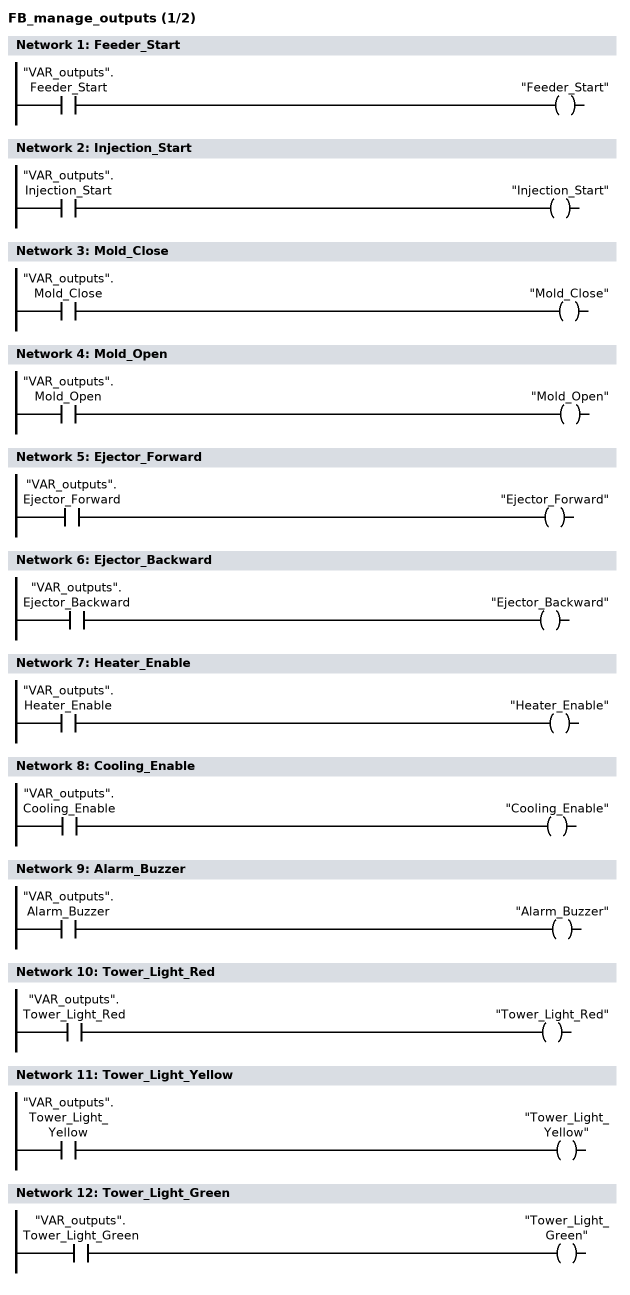
   RUNG wire#powerrail
      Contact( "VAR_outputs".Feeder_Start )
      Coil( "Feeder_Start" )
   END_RUNG
   // the same network as SCL:
   "Feeder_Start" := "VAR_outputs".Feeder_Start;
END_REGION

REGION Network 2: Injection_Start
   RUNG wire#powerrail
      Contact( "VAR_outputs".Injection_Start )
      Coil( "Injection_Start" )
   END_RUNG
   // the same network as SCL:
   "Injection_Start" := "VAR_outputs".Injection_Start;
END_REGION

REGION Network 3: Mold_Close
   RUNG wire#powerrail
      Contact( "VAR_outputs".Mold_Close )
      Coil( "Mold_Close" )
   END_RUNG
   // the same network as SCL:
   "Mold_Close" := "VAR_outputs".Mold_Close;
END_REGION

REGION Network 4: Mold_Open
   RUNG wire#powerrail
      Contact( "VAR_outputs".Mold_Open )
      Coil( "Mold_Open" )
   END_RUNG
   // the same network as SCL:
   "Mold_Open" := "VAR_outputs".Mold_Open;
END_REGION

REGION Network 5: Ejector_Forward
   RUNG wire#powerrail
      Contact( "VAR_outputs".Ejector_Forward )
      Coil( "Ejector_Forward" )
   END_RUNG
   // the same network as SCL:
   "Ejector_Forward" := "VAR_outputs".Ejector_Forward;
END_REGION

REGION Network 6: Ejector_Backward
   RUNG wire#powerrail
      Contact( "VAR_outputs".Ejector_Backward )
      Coil( "Ejector_Backward" )
   END_RUNG
   // the same network as SCL:
   "Ejector_Backward" := "VAR_outputs".Ejector_Backward;
END_REGION

REGION Network 7: Heater_Enable
   RUNG wire#powerrail
      Contact( "VAR_outputs".Heater_Enable )
      Coil( "Heater_Enable" )
   END_RUNG
   // the same network as SCL:
   "Heater_Enable" := "VAR_outputs".Heater_Enable;
END_REGION

REGION Network 8: Cooling_Enable
   RUNG wire#powerrail
      Contact( "VAR_outputs".Cooling_Enable )
      Coil( "Cooling_Enable" )
   END_RUNG
   // the same network as SCL:
   "Cooling_Enable" := "VAR_outputs".Cooling_Enable;
END_REGION

REGION Network 9: Alarm_Buzzer
   RUNG wire#powerrail
      Contact( "VAR_outputs".Alarm_Buzzer )
      Coil( "Alarm_Buzzer" )
   END_RUNG
   // the same network as SCL:
   "Alarm_Buzzer" := "VAR_outputs".Alarm_Buzzer;
END_REGION

REGION Network 10: Tower_Light_Red
   RUNG wire#powerrail
      Contact( "VAR_outputs".Tower_Light_Red )
      Coil( "Tower_Light_Red" )
   END_RUNG
   // the same network as SCL:
   "Tower_Light_Red" := "VAR_outputs".Tower_Light_Red;
END_REGION

REGION Network 11: Tower_Light_Yellow
   RUNG wire#powerrail
      Contact( "VAR_outputs".Tower_Light_Yellow )
      Coil( "Tower_Light_Yellow" )
   END_RUNG
   // the same network as SCL:
   "Tower_Light_Yellow" := "VAR_outputs".Tower_Light_Yellow;
END_REGION

REGION Network 12: Tower_Light_Green
   RUNG wire#powerrail
      Contact( "VAR_outputs".Tower_Light_Green )
      Coil( "Tower_Light_Green" )
   END_RUNG
   // the same network as SCL:
   "Tower_Light_Green" := "VAR_outputs".Tower_Light_Green;
END_REGION

REGION Network 13: Goto_NextStationBuffer
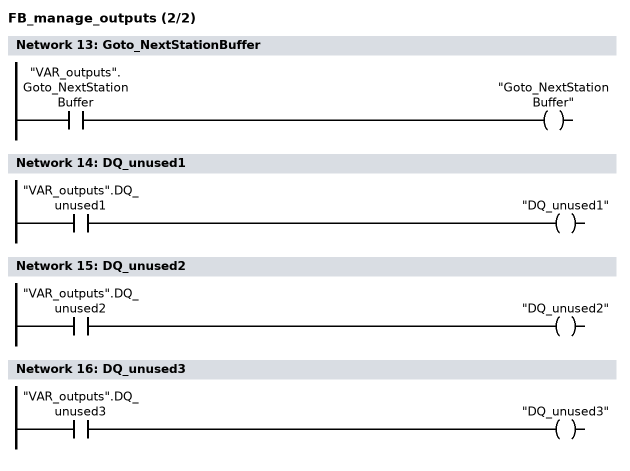
   RUNG wire#powerrail
      Contact( "VAR_outputs".Goto_NextStationBuffer )
      Coil( "Goto_NextStationBuffer" )
   END_RUNG
   // the same network as SCL:
   "Goto_NextStationBuffer" := "VAR_outputs".Goto_NextStationBuffer;
END_REGION

REGION Network 14: DQ_unused1
   RUNG wire#powerrail
      Contact( "VAR_outputs".DQ_unused1 )
      Coil( "DQ_unused1" )
   END_RUNG
   // the same network as SCL:
   "DQ_unused1" := "VAR_outputs".DQ_unused1;
END_REGION

REGION Network 15: DQ_unused2
   RUNG wire#powerrail
      Contact( "VAR_outputs".DQ_unused2 )
      Coil( "DQ_unused2" )
   END_RUNG
   // the same network as SCL:
   "DQ_unused2" := "VAR_outputs".DQ_unused2;
END_REGION

REGION Network 16: DQ_unused3
   RUNG wire#powerrail
      Contact( "VAR_outputs".DQ_unused3 )
      Coil( "DQ_unused3" )
   END_RUNG
   // the same network as SCL:
   "DQ_unused3" := "VAR_outputs".DQ_unused3;
END_REGION
END_FUNCTION_BLOCK

// folder: Simulation_data/Simulation_FB

FUNCTION_BLOCK "FB_simulate_analog_data"   // FB10, LAD
{ S7_Optimized_Access := 'TRUE' }
VERSION : 0.1
   VAR_INPUT
      Clock : Bool;
      Up : Bool;
      Down : Bool;
      TargetLevelLimit : Real;
      HighLevelLimit : Real;
      LowLevelLimit : Real;
      ResetVal : Bool;
   END_VAR
   VAR_IN_OUT
      actLevel : Real;
   END_VAR
   VAR
      value_int : Int;
      value_real : Real;
   END_VAR
   VAR_TEMP
      tag1 : Bool;
   END_VAR
   VAR CONSTANT
      incrementVal : Int := 5;
      decrementVal : Int := 150;
      normMin : Int := 0;
      normMax : Int := 27648;
   END_VAR
   VAR_TEMP   // added for the SCL form of the ladder/FBD networks
      _w1 : Bool;
   END_VAR
BEGIN

REGION Network 1: Simulate an analog input value
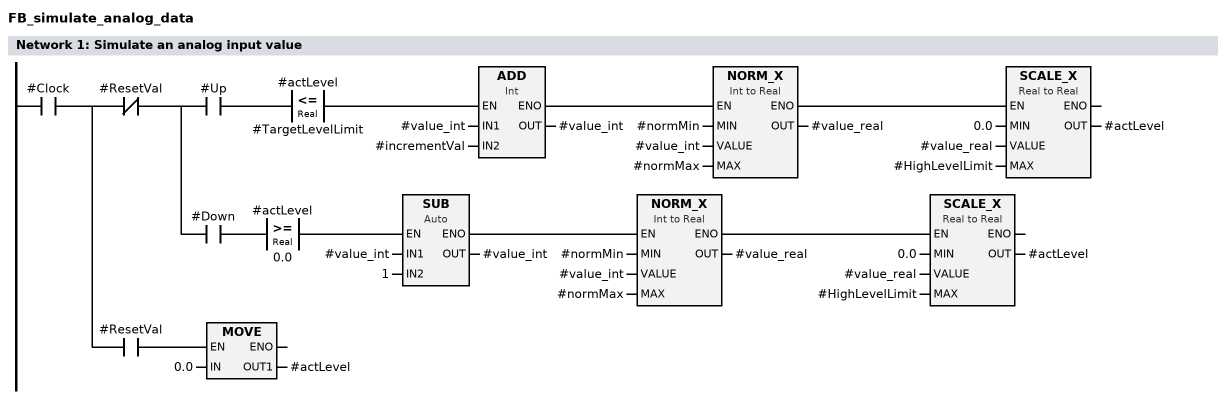
   RUNG wire#powerrail
      Contact( #Clock )
      wire#w1
      I_Contact( #ResetVal )
      wire#w2
      Contact( #Up )
      { S7_Templates := "SrcType := Real" } LE_Contact(in1 := #actLevel, in2 := #TargetLevelLimit)
      { S7_Templates := "SrcType := Int" } Add(in1 := #value_int, in2 := #incrementVal, out => #value_int)
      { S7_Templates := "[SrcType := Int, DestType := Real]" } Normalize(min := #normMin, value := #value_int, max := #normMax, out => #value_real)
      { S7_Templates := "[SrcType := Real, DestType := Real]" } Scale(min := 0.0, value := #value_real, max := #HighLevelLimit, out => #actLevel)
   END_RUNG
   RUNG wire#w2
      Contact( #Down )
      { S7_Templates := "SrcType := Real" } GE_Contact(in1 := #actLevel, in2 := 0.0)
      Sub(in1 := #value_int, in2 := 1, out => #value_int)
      { S7_Templates := "[SrcType := Int, DestType := Real]" } Normalize(min := #normMin, value := #value_int, max := #normMax, out => #value_real)
      { S7_Templates := "[SrcType := Real, DestType := Real]" } Scale(min := 0.0, value := #value_real, max := #HighLevelLimit, out => #actLevel)
   END_RUNG
   RUNG wire#w1
      Contact( #ResetVal )
      Move(in := 0.0, out1 => #actLevel)
   END_RUNG
   // the same network as SCL:
   #_w1 := #Clock AND NOT #ResetVal;
   IF #_w1 AND #Up AND (#actLevel <= #TargetLevelLimit) THEN
       #value_int := #value_int + #incrementVal;
       #value_real := NORM_X(MIN := #normMin, VALUE := #value_int, MAX := #normMax);
       #actLevel := SCALE_X(MIN := 0.0, VALUE := #value_real, MAX := #HighLevelLimit);
   END_IF;
   IF #_w1 AND #Down AND (#actLevel >= 0.0) THEN
       #value_int := #value_int - 1;
       #value_real := NORM_X(MIN := #normMin, VALUE := #value_int, MAX := #normMax);
       #actLevel := SCALE_X(MIN := 0.0, VALUE := #value_real, MAX := #HighLevelLimit);
   END_IF;
   IF #Clock AND #ResetVal THEN #actLevel := 0.0; END_IF;
END_REGION
END_FUNCTION_BLOCK

FUNCTION_BLOCK "FB_simulate_digital_input"   // FB16, LAD
{ S7_Optimized_Access := 'TRUE' }
VERSION : 0.1
   VAR_INPUT
      Open : Bool;
      Close : Bool;
   END_VAR
   VAR_IN_OUT
      Opened : Bool;
      Closed : Bool;
   END_VAR
   VAR
      Sim_timers : Array[0..2] of IEC_TIMER;
   END_VAR
   // Sim_timers[0].PT := T#1S;
   // Sim_timers[1].PT := T#1S;
BEGIN

REGION Network 1
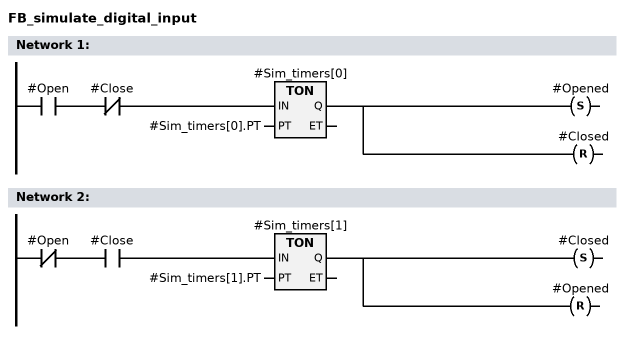
   #Sim_timers[0].TON(IN := #Open AND NOT #Close, PT := #Sim_timers[0].PT);
   IF #Sim_timers[0].Q THEN
       #Opened := TRUE;
       #Closed := FALSE;
   END_IF;
END_REGION

REGION Network 2
   #Sim_timers[1].TON(IN := NOT #Open AND #Close, PT := #Sim_timers[1].PT);
   IF #Sim_timers[1].Q THEN
       #Closed := TRUE;
       #Opened := FALSE;
   END_IF;
END_REGION
END_FUNCTION_BLOCK